// TIA Portal V17 export
// export: Created 2024-06-24T13:41:00.7483362Z, ExportSetting WithDefaults, DisplayName Totally Integrated Automation Portal, DisplayVersion V17, DisplayName TIA Portal Openness, DisplayVersion V17, DisplayName TIA Portal Version Control Interface, DisplayVersion V17, DisplayName STEP 7 Professional, DisplayVersion V17, DisplayName STEP 7 Safety, DisplayVersion V17, DisplayName WinCC Advanced, DisplayVersion V17
ORGANIZATION_BLOCK "Main"   // OB1, LAD, ProgramCycle
TITLE = "Main Program Sweep (Cycle)"
{ S7_Optimized_Access := 'TRUE' }
VERSION : 0.1
// stored: AutoNumber true, IsIECCheckEnabled false, SetENOAutomatically false
   VAR_INPUT
      Initial_Call : Bool;   // Initial call of this OB
      Remanence : Bool;   // =True, if remanent data are available
   END_VAR
BEGIN

REGION Network 1
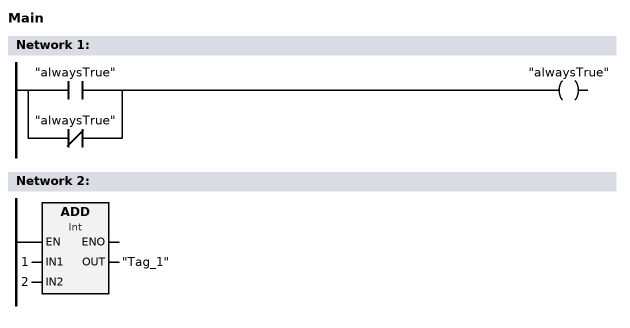
   RUNG wire#powerrail
      Contact( "alwaysTrue" )
      wire#w1
      Coil( "alwaysTrue" )
   END_RUNG
   RUNG wire#powerrail
      I_Contact( "alwaysTrue" )
   END_RUNG wire#w1
   // the same network as SCL:
   "alwaysTrue" := "alwaysTrue" OR NOT "alwaysTrue";
END_REGION

REGION Network 2
   RUNG wire#powerrail
      { S7_Templates := "SrcType := Int" } Add(in1 := 1, in2 := 2, out => "Tag_1")
   END_RUNG
   // the same network as SCL:
   "Tag_1" := 1 + 2;
END_REGION
END_ORGANIZATION_BLOCK
